Fanuc KAREL source: kb00112.KL

-- PROVISIONAL review KL for V1013-1; original PC SHA256 53ea8dfe3200b4f8104f99d9b2ab084d65cc80026ab2cfed58fc52537c3ac1ce
-- Incomplete behavior may be omitted. Consult companion uncertainty JSON. Do not deploy.
PROGRAM KB00112
%NOLOCKGROUP
VAR
  RESULT : BOOLEAN
-- UNRESOLVED_DECL P1 type=000199
BEGIN
  -- UNRESOLVED_PC offsets 5-28; opcodes 27,22,1C,27,9D,76,23
  -- UNRESOLVED_PC offsets 33-37; opcodes 7F
END KB00112
